// TIA Portal V17 export
// export: Created 2024-09-03T21:54:56.2218979Z, ExportSetting WithDefaults, DisplayName Totally Integrated Automation Portal, DisplayVersion V17 Update 7, DisplayName TIA Portal Openness, DisplayVersion V17 Update 7, DisplayName TIA Portal Version Control Interface, DisplayVersion V17, DisplayName SINAMICS Startdrive Advanced, DisplayVersion V17 SP2, DisplayName SINAMICS Startdrive G110M, G120, G120C, G120D, G120P, G115D, DisplayVersion V17 SP2, DisplayName SINAMICS Startdrive G130, G150, S120, S150, SINAMICS MV, S210, DisplayVersion V17 SP2, DisplayName STEP 7 Professional, DisplayVersion V17 Update 7, DisplayName STEP 7 Safety, DisplayVersion V17 Update 6, DisplayName WinCC Advanced / Unified PC, DisplayVersion V17 Update 7
DATA_BLOCK "CycleTimeMeasComplete_DB"   // DB29
VERSION : 0.1
// stored: AutoNumber true, DBAccessibleFromOPCUA true, DBAccessibleFromWebserver true, InstanceOfName CycleTimeMeas, InstanceOfType FB
"CycleTimeMeas"
   // VAR_INPUT
   //    StartCycle : Bool := FALSE;
   //    ResetHistory : Bool := FALSE;
   // END_VAR
   // VAR
   //    ActualTime : Time := T#0MS;
   //    LastTime : Time := T#0MS;
   //    edge2 : Bool := FALSE;
   //    edge1 : Bool := FALSE;
   //    Suma : DInt := 0;
   //    Count : DInt := 0;
   //    Max : Time := T#0MS;
   //    Min : Time := T#0MS;
   //    Average : Time := T#0MS;
   //    IEC_Timer_0_Instance { S7_SetPoint := 'True'} : TON_TIME;
   //    History : Array[1..20] of Time;
   //    NewTime : Bool := FALSE;
   // END_VAR
BEGIN
   IEC_Timer_0_Instance.PT := T#0MS;
   IEC_Timer_0_Instance.IN := FALSE;
   History[1..20] := T#0MS;
END_DATA_BLOCK
